(*Electrical device with continous operation mode*)
TYPE ElectrDeviceContOper_DataModel :
STRUCT
	LineName	: STRING(40);
	MachineName	: STRING(40);
	DeviceName	: STRING(40);
	
	ElectricalData : ElectrDataModbusTCP;
	
	TimeStamp 	: ULINT;
END_STRUCT
END_TYPE

(* stored: Version 1.1.0.1, ProductVersion 3.1.4024.15
   DUT ElectrDeviceContOper_DataModel: Id {39274b22-511f-40b5-86e5-5fdcf09753dd} *)
